FUNCTION_BLOCK verticalcylinder3 (* Basic Function Block Type *)
  (* Standard: 61499-2 *)
  (* Version 0.0, 2011-02-26, Majid Sorouri, nxtControl GmbH, Template *)
  (* Compiler header: package fb.rt.pnp; *)
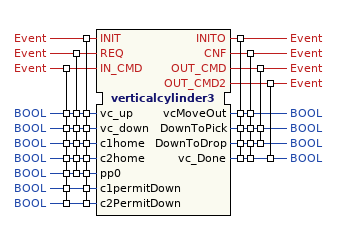
  EVENT_INPUT
    INIT WITH vc_up, vc_down, c1home, c2home, pp0, c1permitDown, c2PermitDown; (* Initialization Request *)
    REQ WITH vc_up, vc_down, c1home, c2home, pp0; (* Normal Execution Request *)
    IN_CMD WITH c1permitDown, vc_up, vc_down, c1home, c2home, pp0, c2PermitDown;
  END_EVENT
  EVENT_OUTPUT
    INITO WITH DownToPick, DownToDrop, vc_Done, vcMoveOut; (* Initialization Confirm *)
    CNF WITH vcMoveOut, DownToPick, DownToDrop, vc_Done;
    OUT_CMD WITH DownToPick, DownToDrop;
    OUT_CMD2 WITH vc_Done;
  END_EVENT
  VAR_INPUT
    vc_up : BOOL; (* Input event qualifier *)
    vc_down : BOOL;
    c1home : BOOL;
    c2home : BOOL;
    pp0 : BOOL;
    c1permitDown : BOOL;
    c2PermitDown : BOOL;
  END_VAR
  VAR_OUTPUT
    vcMoveOut : BOOL; (* Output event qualifier *)
    DownToPick : BOOL;
    DownToDrop : BOOL;
    vc_Done : BOOL;
  END_VAR
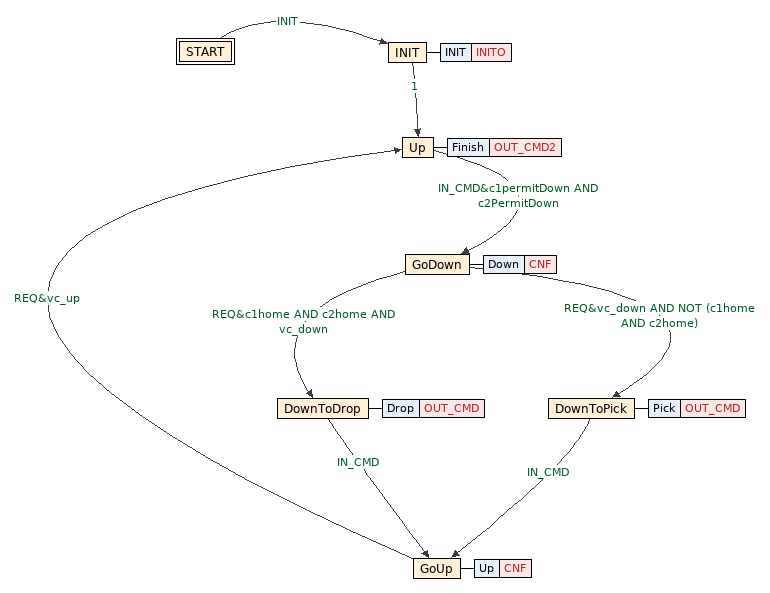
  EC_STATES
    START; (* Initial State *)
    INIT : INIT -> INITO; (* Initialization *)
    GoUp : Up -> CNF;
    GoDown : Down -> CNF;
    DownToPick : Pick -> OUT_CMD;
    DownToDrop : Drop -> OUT_CMD;
    Up : Finish -> OUT_CMD2;
  END_STATES
  EC_TRANSITIONS
    START TO INIT := INIT;
    DownToDrop TO GoUp := IN_CMD;
    GoDown TO DownToPick := REQ&vc_down AND NOT (c1home AND c2home);
    GoDown TO DownToDrop := REQ&c1home AND c2home AND vc_down;
    GoUp TO Up := REQ&vc_up;
    DownToPick TO GoUp := IN_CMD;
    Up TO GoDown := IN_CMD&c1permitDown AND c2PermitDown;
    INIT TO Up := 1;
  END_TRANSITIONS
  ALGORITHM INIT IN ST: (* Initialization algorithm *)
vcMoveOut:=FALSE;
DownToPick:=FALSE;
DownToDrop:=FALSE;
vc_Done:=TRUE;
System.out.println("VertCyl INIT");
  END_ALGORITHM
  ALGORITHM Down IN ST:
vcMoveOut:=TRUE;
vc_Done:=FALSE;
System.out.println("VertCyl Down");
  END_ALGORITHM
  ALGORITHM Up IN ST:
vcMoveOut:=FALSE;
System.out.println("VertCyl Up");
  END_ALGORITHM
  ALGORITHM Pick IN ST:
DownToPick:=TRUE;
DownToDrop:=FALSE;
System.out.println("VertCyl Pick");
  END_ALGORITHM
  ALGORITHM Drop IN ST:
DownToPick:=FALSE;
DownToDrop:=TRUE;
System.out.println("VertCyl Drop");
  END_ALGORITHM
  ALGORITHM Finish IN ST:
vc_Done:=TRUE;
System.out.println("VertCyl Finish");
  END_ALGORITHM
END_FUNCTION_BLOCK
